FUNCTION_BLOCK FB_SingleTank
VAR
	sName : STRING;
	sWeightUnit : STRING := 'Kg'; // Kg
	piLslow : FB_DigitalInput;
	piLsHigh : FB_DigitalInput;
	poCylinderCoil : FB_DigitalOutput;
END_VAR

PROPERTY Name : String
GET
Name := sName;
END_GET
SET
sName := Name;
END_SET
END_PROPERTY

PROPERTY Ref_piLsHigh : reference to FB_DigitalInput
GET
Ref_piLsHigh ref= piLsHigh;
END_GET
END_PROPERTY

PROPERTY Ref_piLsLow : reference to FB_DigitalInput
GET
Ref_piLsLow ref= piLslow;
END_GET
END_PROPERTY

PROPERTY Ref_poCylinderCoil : REFERENCE TO FB_DigitalOutput
GET
Ref_poCylinderCoil ref= poCylinderCoil;
END_GET
END_PROPERTY

PROPERTY WeightUnit : string
GET
WeightUnit := sWeightUnit;
END_GET
SET
sWeightUnit := WeightUnit;
END_SET
END_PROPERTY

END_FUNCTION_BLOCK

(* stored: Version 1.1.0.1, ProductVersion 3.1.4024.12
   POU FB_SingleTank: Id {fb97367d-7b47-44e9-8c40-eeee1f05ceee}, SpecialFunc None
   Property Name: Id {a7647dce-070a-425b-99fc-11d432804333}
   Get Get: Id {dd3fac2e-05af-4186-a43b-0d03e88b709e}
   Set Set: Id {2be577ed-204f-4885-9934-5c2ffce1c9a1}
   Property Ref_piLsHigh: Id {7e7f4737-2362-4583-a3a2-cd6dfee5ec62}
   Get Get: Id {19e0dff5-6a0e-44b0-9293-2f2309385d1b}
   Property Ref_piLsLow: Id {602bc692-fbb2-4ec7-a243-8b8e8ee96c4d}
   Get Get: Id {450a7dc7-f7f5-45a6-abbc-8937ab6a5af5}
   Property Ref_poCylinderCoil: Id {e609a428-6ab3-40cb-a686-885573c121fa}
   Get Get: Id {4ac1a50a-33c2-4df0-bdef-7dc65bbb0f72}
   Property WeightUnit: Id {77dbb17f-7210-4007-b0ad-d8ccfe7a3644}
   Get Get: Id {238a38ad-a707-4a80-8507-4f57900189f0}
   Set Set: Id {522630ab-9f84-43ad-a730-dd4797fe41d8} *)
